// TIA Portal V16 export
// export: Created 2023-08-28T09:37:54.7506472Z, ExportSetting WithDefaults, DisplayName Totally Integrated Automation Portal, DisplayVersion V16 Update 6, DisplayName TIA Portal Version Control Interface, DisplayVersion V16 Update 2, DisplayName TIA Portal Openness, DisplayVersion V16 Update 6, DisplayName STEP 7 Professional, DisplayVersion V16 Update 6, DisplayName STEP 7 Safety, DisplayVersion V16, DisplayName WinCC Advanced, DisplayVersion V16 Update 6
VAR_GLOBAL   // PLC tag table "Analogs"
   IW68 AT %IW68 : Int;
   IW66 AT %IW66 : Int;
   IW64 AT %IW64 : Int;
   IW70 AT %IW70 : Int;
   switch_kolman AT %M18.7 : Bool;   // załącz/ wyłą filtrowanie przez kolmana analogów
   "i(1)" AT %MW112 : Int;
END_VAR
